# EPICS SNL sequencer program: apps/svtCtrlApp/src/seq_svtOnOff.st
program seq_test

option -c;
option -r;
option -s;

%%#include <stdlib.h>

#define NREGIONS 4
#define NCHANS 96
#define NSIDES 2
#define NANADIG 2

string prefix="B_SVT";
string hv_vmonSuff=":outputMeasSenseV";
string lv_vmonSuff=":outputMeasSenseV";
string hv_switchSuff=":outSwitch";
string lv_switchSuff=":onOff";

string sides[NSIDES]={"T","B"};
string anadig[NANADIG]={"A","D"};

int nModulesPerRegion[NREGIONS]={10,14,18,24};
int hv_slotsPerRegion[NREGIONS][4]={ { 7,8,9,10}, { 9,10,0,0}, { 8, 9,10,0}, { 8, 9,10,0} };
int hv_nChansPerSlot[NREGIONS][4] ={ {16,4,0, 0}, {16,12,0,0}, {16,16, 4,0}, {16,16,16,0} };

#define NPVSTATIC 7
string msg;    assign msg      to "B_SVT_R{R}_SEQ:msg";
short btnOff;  assign btnOff   to "B_SVT_R{R}_SEQ:btnOff";  monitor btnOff;
short btnOn;   assign btnOn    to "B_SVT_R{R}_SEQ:btnOn";   monitor btnOn;
int lv_isOn;   assign lv_isOn  to "B_SVT_LV_R{R}:isOn";     monitor lv_isOn;
int lv_isOff;  assign lv_isOff to "B_SVT_LV_R{R}:isOff";    monitor lv_isOff;
int hv_isOn;   assign hv_isOn  to "B_SVT_HV_R{R}:isOn";     monitor hv_isOn;
int hv_isOff;  assign hv_isOff to "B_SVT_HV_R{R}:isOff";    monitor hv_isOff;
//int watchdog;  assign watchdog to "B_SVT_R{R}_SEQ:heartbeat";

double hv_vmon[NCHANS]; assign hv_vmon to {};
double lv_vmon[NCHANS]; assign lv_vmon to {};
int hv_switch[NCHANS];  assign hv_switch to {};
int lv_switch[NCHANS];  assign lv_switch to {};

string stmp;
string stub;
string sRegion;
int hv_nChan=0;
int lv_nChan=0;
int hv_iSlot;
int hv_nChanSlot;
int nPVs=0;
int ii,jj,kk;
int slot;
int iRegion;
int exitError=0;

ss seq_test {

    state start {

        entry {
            nPVs = NPVSTATIC;
            sprintf(sRegion,"%s",macValueGet("R"));
            sprintf(stub,"seq_test(%s)",sRegion);
            if (strcmp(sRegion,"1")!=0 &&
                strcmp(sRegion,"2")!=0 &&
                strcmp(sRegion,"3")!=0 &&
                strcmp(sRegion,"4")) {
                exitError=1;
                sprintf(msg,"start: Invalid Region (%s), EXITING.",sRegion);
                printf("\n%s - %s\n\n",stub,msg);
                pvPut(msg);
            }
            iRegion=atoi(sRegion);
        }

        when (exitError) {} exit

        when (pvConnectCount() < nPVs) {
            sprintf(msg,"start: Waiting for PVs (%d/%d)",pvConnectCount(),nPVs);
            printf("\n%s - %s\n\n",stub,msg);
            pvPut(msg);
            epicsThreadSleep(1);
        } state start

        when () {} state init
    }

    state init {

        entry {
            sprintf(msg,"init: Assigning PVs ...");
            printf("\n%s - %s\n\n",stub,msg);
            pvPut(msg);
            hv_nChan=0;
            lv_nChan=0;
            hv_iSlot=0;
            hv_nChanSlot=0;
            for (ii=0; ii<nModulesPerRegion[iRegion-1]; ii++) {

                for (jj=0; jj<NSIDES; jj++) {

                    // HV:
                    // slot mapping defined by global arrays above
                    slot = hv_slotsPerRegion[iRegion-1][hv_iSlot];
                    sprintf(stmp,"%s_HV_R%dS%d%s_Slot%d%s",prefix,
                            iRegion,ii+1,sides[jj],slot,hv_vmonSuff);
                    pvAssign(hv_vmon[hv_nChan],stmp);
                    sprintf(stmp,"%s_HV_R%dS%d%s_Slot%d%s",prefix,
                            iRegion,ii+1,sides[jj],slot,hv_switchSuff);
                    pvAssign(hv_switch[hv_nChan],stmp);
                    hv_nChan++;
                    nPVs += 2;

                    // LV:
                    // slot mapping just starts at 1, with 8 channels per slot,
                    // except R4 starts over after Slot6
                    for (kk=0; kk<NANADIG; kk++) {
                        slot = (ii*4+jj*2+kk)/8+1;
                        if (iRegion==4 && slot>6) slot-=6;
                        sprintf(stmp,"%s_LV_V%s_R%dS%d%s_Slot%d%s",prefix,
                                anadig[kk],iRegion,ii+1,sides[jj],slot,lv_vmonSuff);
                        pvAssign(lv_vmon[lv_nChan],stmp);
                        sprintf(stmp,"%s_LV_V%s_R%dS%d%s_Slot%d%s",prefix,
                                anadig[kk],iRegion,ii+1,sides[jj],slot,lv_switchSuff);
                        pvAssign(lv_switch[lv_nChan],stmp);
                        lv_nChan++;
                        nPVs += 2;
                    }
                }

                hv_nChanSlot += 2;
                if (hv_nChanSlot >= hv_nChansPerSlot[iRegion-1][hv_iSlot])
                {
                    hv_iSlot++;
                    hv_nChanSlot=0;
                }
            }
        }

        when (pvConnectCount() < nPVs) {
            sprintf(msg,"init: Waiting for PVs (%d/%d)",pvConnectCount(),nPVs);
            printf("\n%s - %s\n\n",stub,msg);
            pvPut(msg);
            epicsThreadSleep(2);
        } state listen
    }

    state listen {
        entry {
            sprintf(msg,"Waiting for Signal ...");
            printf("\n%s - %s\n\n",stub,msg);
            pvPut(msg);
        }
        when (pvConnectCount() < nPVs) {
            sprintf(msg,"listen: Waiting for PVs (%d/%d)",pvConnectCount(),nPVs);
            printf("\n%s - %s\n\n",stub,msg);
            pvPut(msg);
            epicsThreadSleep(2);
        } state listen
        when (btnOff) {
            btnOff=0;
            pvPut(btnOff);
        } state hvoff
        when (btnOn) {
            btnOn=0;
            pvPut(btnOn);
        } state lvon
        when () {
            epicsThreadSleep(1);
        } state listen
    }

    // listen -> lvon -> hvon -> listen
    // listen -> hvoff -> lvoff -> listen

    state lvon {
        entry {
            sprintf(msg,"lvon ...");
            printf("\n%s - %s\n\n",stub,msg);
            pvPut(msg);
            for (ii=0; ii<lv_nChan; ii++) {
                printf("%d\n",ii);
                //lv_switch[jj]=1;
                //pvPut(lv_switch[jj]);
                if ((ii+1)%10==0) epicsThreadSleep(1);
            }
        }
        when (btnOff) {
            btnOff=0;
            pvPut(btnOff);
        } state hvoff
        when (btnOn) {
            btnOn=0;
            pvPut(btnOn);
        } state lvon
        when (lv_isOn) {} state hvon
    }

    state hvon {
        entry {
            sprintf(msg,"hvon ...");
            printf("\n%s - %s\n\n",stub,msg);
            pvPut(msg);
            for (ii=0; ii<hv_nChan; ii++) {
                printf("%d\n",ii);
                //hv_switch[jj]=1;
                //pvPut(hv_switch[jj]);
                if ((ii+1)%10==0) epicsThreadSleep(1);
            }
        }
        when (btnOff) {
            btnOff=0;
            pvPut(btnOff);
        } state hvoff
        when (btnOn) {
            btnOn=0;
            pvPut(btnOn);
        } state hvon
        when (hv_isOn) {
        } state listen

    }

    state hvoff {
        entry {
            sprintf(msg,"hvoff ...");
            printf("\n%s - %s\n\n",stub,msg);
            pvPut(msg);
            for (ii=0; ii<hv_nChan; ii++) {
                printf("%d\n",ii);
                //hv_switch[jj]=0;
                //pvPut(hv_switch[jj]);
                if ((ii+1)%10==0) epicsThreadSleep(1);
            }
        }
        when (btnOff) {
            btnOff=0;
            pvPut(btnOff);
        } state hvoff
        when (btnOn) {
            btnOn=0;
            pvPut(btnOn);
        } state lvon
        when (hv_isOff) {} state lvoff
    }

    state lvoff {
        entry {
            sprintf(msg,"lvoff ...");
            printf("\n%s - %s\n\n",stub,msg);
            pvPut(msg);
            for (ii=0; ii<lv_nChan; ii++) {
                printf("%d\n",ii);
                //lv_switch[jj]=0;
                //pvPut(lv_switch[jj]);
                if ((ii+1)%10==0) epicsThreadSleep(1);
            }
        }
        when (btnOff) {
            btnOff=0;
            pvPut(btnOff);
        } state lvoff
        when (btnOn) {
            btnOn=0;
            pvPut(btnOn);
        } state lvon
        when (lv_isOff) {} state listen
    }

}
